Staubli VAL3: getStatusWord.pgx

public program getStatusWord(num x_nAxisNumber, num& x_nValue)
begin
  // this routine return the value of the drive's status word
  //
  x_nValue=aioGet(aiStatusWord[x_nAxisNumber])
end
